// TIA Portal V18 export
TYPE "UDT_AObasic"
// stored: IsFailsafeCompliant false
   STRUCT
      iID : DInt;   // AOs ID for monitoring
      rInput : Real;   // Value for AO
      cMOA : Byte;   // Mode Manual/Off/Auto
      rMan_output : Real;   // Manual output
      iOutput : Int;   // Output for DAC
      wMark : String["IOmark_string_length"];   // AOs label for monitoring
   END_STRUCT;
END_TYPE
